TYPE ST_TxHmiWinch :
STRUCT
	status : DINT := 0;
	l : REAL; 
	l_t : REAL;
	l_tt : REAL;
END_STRUCT
END_TYPE

(* stored: Version 1.1.0.1, ProductVersion 3.1.4022.7
   DUT ST_TxHmiWinch: Id {ae894732-388f-49a5-a442-5bb07b53ffa7} *)
